FUNCTION_BLOCK Pre_Tratamento (* Composite Function Block Type *)
  (* Standard: 61499-2 *)
  (* Version 0.0, 09/03/2026, template *)
  PACKAGE Hidryco.HidrycoLib;
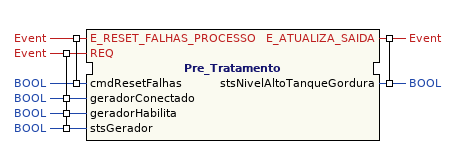
  EVENT_INPUT
    E_RESET_FALHAS_PROCESSO WITH cmdResetFalhas;
    REQ WITH geradorConectado, geradorHabilita, stsGerador;
  END_EVENT
  EVENT_OUTPUT
    E_ATUALIZA_SAIDA WITH stsNivelAltoTanqueGordura;
  END_EVENT
  VAR_INPUT
    cmdResetFalhas : BOOL;
    geradorConectado : BOOL;
    geradorHabilita : BOOL;
    stsGerador : BOOL;
  END_VAR
  VAR_OUTPUT
    stsNivelAltoTanqueGordura : BOOL;
  END_VAR
  FBS
    Peneira_Rotativa1 : Peneira_Rotativa;
    Compressor1 : Compressor;
    Rosca1Horizontal : Rosca;
    Rosca2Inclinada : Rosca;
    Raspador_Gordura1 : Raspador_Gordura;
    SYMLINKMULTIVARDST1 : SYMLINKMULTIVARDST_173DE751D51121F49(NAME1 := '$${PATH}stsEmergenciaAcionada', NAME2 := '$${PATH}stsNivelBaixoPeneira', NAME3 := '$${PATH}stsNivelAltoPeneira', NAME4 := '$${PATH}stsNivelBaixoTanqueAgua', NAME5 := '$${PATH}stsNivelAltoTanqueGordura', NAME6 := '$${PATH}stsNivelPeneira', QI := TRUE); {SET_ATTRIBUTE(Configuration.GenericFBType.InterfaceParams, Runtime.System#I:=6;VALUE${I$}:BOOL,BOOL,BOOL,BOOL,BOOL,INT)}
    IThis : Pre_Tratamento_HMI(QI := TRUE);
    SYMLINKMULTIVARSRC1 : SYMLINKMULTIVARSRC_91EC7219ED37E472(QI := TRUE, NAME1 := '$${PATH}cmdLigaSubsistemaPeneira', NAME2 := '$${PATH}cmdSelecaoSubsistemaPeneira', NAME3 := '$${PATH}cmdLigaSubsistemaRoscas', NAME4 := '$${PATH}cmdLigaSelecaoSubsistemaRoscas', NAME5 := '$${PATH}cmdLigaSubsistemaRaspComp', NAME6 := '$${PATH}cmdSelecaoSubsistemaRaspComp', NAME7 := '$${PATH}cmdSelecaoBombaHigienizacao', NAME8 := '$${PATH}cmdResetPainel'); {SET_ATTRIBUTE(Configuration.GenericFBType.InterfaceParams, Runtime.System#I:=8;VALUE${I$}:BOOL,BOOL,BOOL,BOOL,BOOL,BOOL,BOOL,BOOL)}
    plcStart1 : plcStart(Prio := 10);
    Bomba_Higienizacao1 : Bomba_Higienizacao;
    Bomba_Higienizacao2 : Bomba_Higienizacao;
    Valvula_Higienizacao1 : Valvula_Higienizacao;
    Valvula_Higienizacao2 : Valvula_Higienizacao;
    E_MERGE1 : E_MERGE;
    OR1 : OR_148CCC6046D4CE74C; {SET_ATTRIBUTE(Configuration.GenericFBType.InterfaceParams, Runtime.Standard#CNT:=2)}
    animacao_icone_gerador1 : animacao_icone_gerador;
    COMPARE1 : COMPARE_739E3FB559152FE(IN2 := 1); {SET_ATTRIBUTE(Configuration.GenericFBType.InterfaceParams, Runtime.Standard#CNT:=2;IN${CNT$}:INT)}
  END_FBS
  EVENT_CONNECTIONS
    plcStart1.REDO_INIT TO SYMLINKMULTIVARDST1.INIT;
    plcStart1.FIRST_INIT TO SYMLINKMULTIVARDST1.INIT;
    SYMLINKMULTIVARSRC1.INITO TO plcStart1.ACK_FIRST;
    Bomba_Higienizacao2.E_ATUALIZA_ANIMACAO TO E_MERGE1.EI1;
    Valvula_Higienizacao2.E_ATUALIZA_ANIMACAO TO E_MERGE1.EI1;
    Raspador_Gordura1.E_ATUALIZA_ANIMACAO TO E_MERGE1.EI1;
    Compressor1.E_ATUALIZA_ANIMACAO TO E_MERGE1.EI1;
    Rosca1Horizontal.E_ATUALIZA_ANIMACAO TO E_MERGE1.EI1;
    Rosca2Inclinada.E_ATUALIZA_ANIMACAO TO E_MERGE1.EI1;
    Peneira_Rotativa1.E_ATUALIZA_ANIMACAO TO E_MERGE1.EI1;
    Bomba_Higienizacao1.E_ATUALIZA_ANIMACAO TO E_MERGE1.EI1;
    Valvula_Higienizacao1.E_ATUALIZA_ANIMACAO TO E_MERGE1.EI1;
    SYMLINKMULTIVARDST1.CNF TO E_ATUALIZA_SAIDA;
    E_RESET_FALHAS_PROCESSO TO OR1.REQ;
    OR1.CNF TO SYMLINKMULTIVARSRC1.REQ;
    SYMLINKMULTIVARDST1.INITO TO IThis.73379897072C99BC;
    SYMLINKMULTIVARDST1.CNF TO IThis.AB568CC2EE3C6987;
    SYMLINKMULTIVARDST1.CNF TO IThis.74D389496A49EC77;
    E_MERGE1.EO TO IThis.74D389496A49EC77;
    IThis.94C460257F7023C6 TO SYMLINKMULTIVARSRC1.INIT;
    IThis.E8AF34262A3C4689 TO SYMLINKMULTIVARSRC1.REQ;
    IThis.E8AF34262A3C4689 TO Peneira_Rotativa1.E_ATUALIZA_SUBSISTEMA;
    IThis.E8AF34262A3C4689 TO Valvula_Higienizacao2.E_ATUALIZA_SUBSISTEMA;
    IThis.E8AF34262A3C4689 TO Bomba_Higienizacao2.E_ATUALIZA_SUBSISTEMA;
    IThis.E8AF34262A3C4689 TO Bomba_Higienizacao1.E_ATUALIZA_SUBSISTEMA;
    IThis.E8AF34262A3C4689 TO Valvula_Higienizacao1.E_ATUALIZA_SUBSISTEMA;
    IThis.E8AF34262A3C4689 TO Rosca1Horizontal.E_ATUALIZA_SUBSISTEMA;
    IThis.E8AF34262A3C4689 TO Rosca2Inclinada.E_ATUALIZA_SUBSISTEMA;
    IThis.E8AF34262A3C4689 TO Compressor1.E_ATUALIZA_SUBSISTEMA;
    IThis.E8AF34262A3C4689 TO Raspador_Gordura1.E_ATUALIZA_SUBSISTEMA;
    IThis.9F72FDD749D51B8C TO OR1.REQ;
    Peneira_Rotativa1.E_ATUALIZA_ANIMACAO TO COMPARE1.REQ;
    COMPARE1.CNF TO animacao_icone_gerador1.6664704A75AB52C7;
    REQ TO animacao_icone_gerador1.6664704A75AB52C7;
  END_CONNECTIONS
  DATA_CONNECTIONS
    SYMLINKMULTIVARDST1.VALUE5 TO stsNivelAltoTanqueGordura;
    cmdResetFalhas TO OR1.IN1;
    OR1.OUT TO SYMLINKMULTIVARSRC1.VALUE8;
    SYMLINKMULTIVARDST1.VALUE1 TO IThis.344F99B3F221DB89;
    SYMLINKMULTIVARDST1.VALUE2 TO IThis.206D2400C77475EC;
    SYMLINKMULTIVARDST1.VALUE3 TO IThis.F741E4CC87E9D360;
    SYMLINKMULTIVARDST1.VALUE4 TO IThis.D4295186230E03C6;
    SYMLINKMULTIVARDST1.VALUE5 TO IThis.56CF445F3EE52492;
    SYMLINKMULTIVARDST1.VALUE6 TO IThis.2F6D2B97D6A00BFD;
    Bomba_Higienizacao1.stsAnimacao TO IThis.57041474E7AFFD48;
    Bomba_Higienizacao2.stsAnimacao TO IThis.A2A9C8927C23787B;
    Peneira_Rotativa1.stsAnimacao TO IThis.227C498FDB5AF3BC;
    Valvula_Higienizacao1.stsAnimacao TO IThis.474889046A548AE8;
    Valvula_Higienizacao2.stsAnimacao TO IThis.1F6E3D562A459F84;
    Compressor1.stsAnimacao TO IThis.58544991851041D9;
    Raspador_Gordura1.stsAnimacao TO IThis.8342CB3B4DD198F8;
    Rosca1Horizontal.stsAnimacao TO IThis.8375DF01E23091AE;
    Rosca2Inclinada.stsAnimacao TO IThis.4E8B75A16AE36159;
    animacao_icone_gerador1.9C79DED157DD322B TO IThis.2E2B3C3157EA553A;
    IThis.D555435FD54ACD9C TO SYMLINKMULTIVARSRC1.VALUE1;
    IThis.E2BEA107859CE40F TO SYMLINKMULTIVARSRC1.VALUE2;
    IThis.E2BEA107859CE40F TO Bomba_Higienizacao2.stsAutomaticoSubsistema;
    IThis.E2BEA107859CE40F TO Valvula_Higienizacao2.stsAutomaticoSubsistema;
    IThis.E2BEA107859CE40F TO Bomba_Higienizacao1.stsAutomaticoSubsistema;
    IThis.E2BEA107859CE40F TO Valvula_Higienizacao1.stsAutomaticoSubsistema;
    IThis.E2BEA107859CE40F TO Peneira_Rotativa1.stsAutomaticoSubsistema;
    IThis.DE8C26FB35029C35 TO SYMLINKMULTIVARSRC1.VALUE3;
    IThis.7CF47BAFC9419307 TO SYMLINKMULTIVARSRC1.VALUE4;
    IThis.7CF47BAFC9419307 TO Rosca1Horizontal.stsAutomaticoSubsistema;
    IThis.7CF47BAFC9419307 TO Rosca2Inclinada.stsAutomaticoSubsistema;
    IThis.D14ACEFD049ED51A TO SYMLINKMULTIVARSRC1.VALUE5;
    IThis.470EBB1A8DC6B25 TO SYMLINKMULTIVARSRC1.VALUE6;
    IThis.470EBB1A8DC6B25 TO Compressor1.stsAutomaticoSubsistema;
    IThis.470EBB1A8DC6B25 TO Raspador_Gordura1.stsAutomaticoSubsistema;
    IThis.D49E6658FAC6CE84 TO SYMLINKMULTIVARSRC1.VALUE7;
    IThis.43DDB15809461D8D TO OR1.IN2;
    Peneira_Rotativa1.stsAnimacao TO COMPARE1.IN1;
    COMPARE1.EQ TO animacao_icone_gerador1.9BDA490118C2DB82;
    stsGerador TO animacao_icone_gerador1.D1F24EEF47EA35FE;
    geradorConectado TO animacao_icone_gerador1.3423BEAECBF17FFD;
    geradorHabilita TO animacao_icone_gerador1.D7467A745E6CDBA8;
  END_CONNECTIONS
END_FUNCTION_BLOCK
